% RSLogix 500 project P2_ABIOLA_A_TESTING V7.RSS, saved by version 8.30.00.16 %
PROJECT "UNTITLED"    % processor: Bul.1763 MicroLogix 1100 Series B %

PROGRAM FILES
  LAD 2   4 rungs
  LAD 3 "INPUT DVS"  5 rungs  % This contains all the input devices used %
  LAD 4 "OUTPUT DVS"  4 rungs  % This contains all the output device used %
  LAD 5 "PRO LOGIC"  6 rungs  % This contains the implementation of the logic %

DATA FILES
  O0 OUTPUT  4 elements
  I1 INPUT  6 elements
  S2 STATUS  66 elements
  B3 BINARY  1 elements
  T4 TIMER  2 elements
  C5 COUNTER  1 elements
  R6 CONTROL  1 elements
  N7 INTEGER  1 elements
  F8 FLOAT  1 elements

LADDER 2
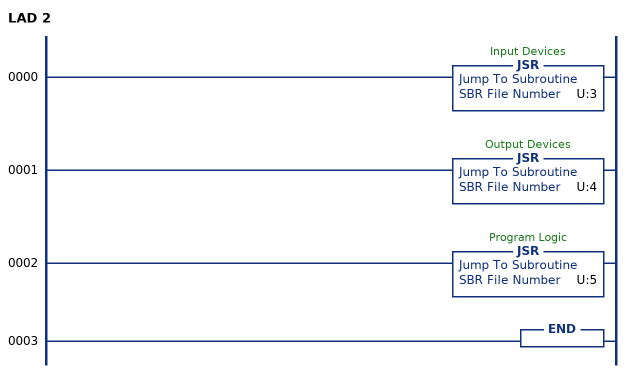
% Rung: 0 %
SOR JSR U:3 EOR
%   U:3  "Input Devices" %
% Rung: 1 %
SOR JSR U:4 EOR
%   U:4  "Output Devices" %
% Rung: 2 %
SOR JSR U:5 EOR
%   U:5  "Program Logic" %
% Rung: 3 %
SOR END EOR

LADDER 3 "INPUT DVS"    % This contains all the input devices used %
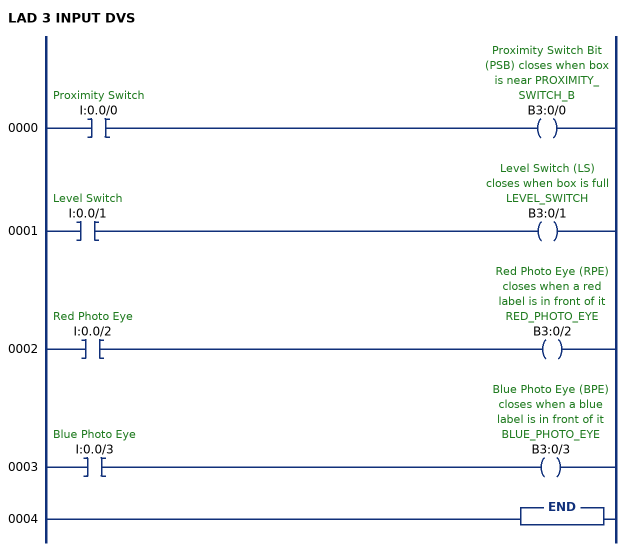
% Rung: 0 %
SOR XIC I:0.0/0 OTE B3:0/0 EOR
%   I:0.0/0  "Proximity Switch" %
%   B3:0/0  PROXIMITY_SWITCH_B  "Proximity Switch Bit (PSB) closes when box is near" %
% Rung: 1 %
SOR XIC I:0.0/1 OTE B3:0/1 EOR
%   I:0.0/1  "Level Switch" %
%   B3:0/1  LEVEL_SWITCH  "Level Switch (LS) closes when box is full" %
% Rung: 2 %
SOR XIC I:0.0/2 OTE B3:0/2 EOR
%   I:0.0/2  "Red Photo Eye" %
%   B3:0/2  RED_PHOTO_EYE  "Red Photo Eye (RPE) closes when a red label is in front of it" %
% Rung: 3 %
SOR XIC I:0.0/3 OTE B3:0/3 EOR
%   I:0.0/3  "Blue Photo Eye" %
%   B3:0/3  BLUE_PHOTO_EYE  "Blue Photo Eye (BPE) closes when a blue label is in front of it" %
% Rung: 4 %
SOR END EOR

LADDER 4 "OUTPUT DVS"    % This contains all the output device used %
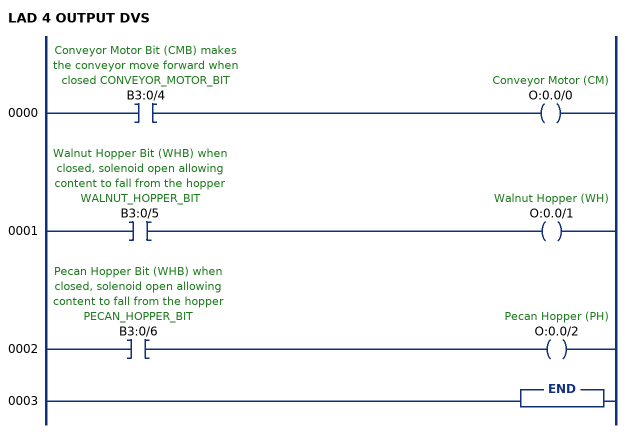
% Rung: 0 %
SOR XIC B3:0/4 OTE O:0.0/0 EOR
%   B3:0/4  CONVEYOR_MOTOR_BIT  "Conveyor Motor Bit (CMB) makes the conveyor move forward when closed" %
%   O:0.0/0  "Conveyor Motor (CM)" %
% Rung: 1 %
SOR XIC B3:0/5 OTE O:0.0/1 EOR
%   B3:0/5  WALNUT_HOPPER_BIT  "Walnut Hopper Bit (WHB) when closed, solenoid open allowing content to fall from the hopper" %
%   O:0.0/1  "Walnut Hopper (WH)" %
% Rung: 2 %
SOR XIC B3:0/6 OTE O:0.0/2 EOR
%   B3:0/6  PECAN_HOPPER_BIT  "Pecan Hopper Bit (WHB) when closed, solenoid open allowing content to fall from the hopper" %
%   O:0.0/2  "Pecan Hopper (PH)" %
% Rung: 3 %
SOR END EOR

LADDER 5 "PRO LOGIC"    % This contains the implementation of the logic %
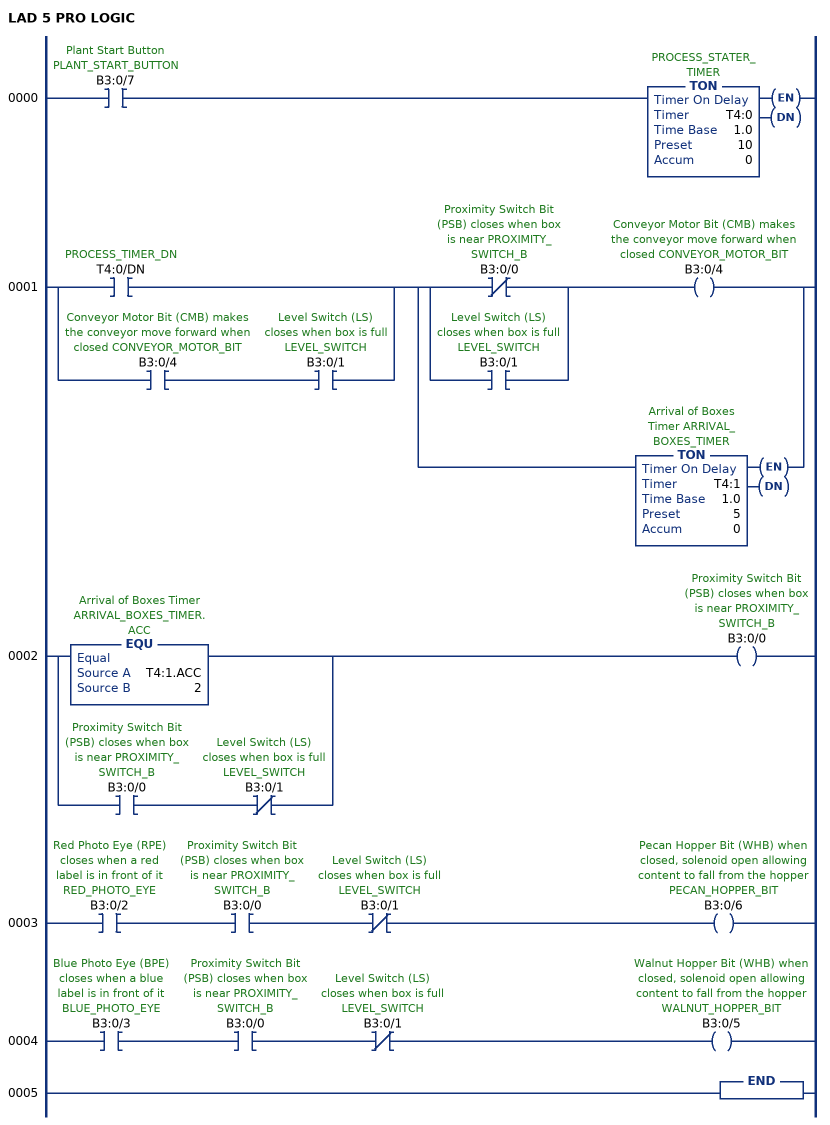
% Rung: 0 %
SOR XIC B3:0/7 TON T4:0 1.0 10 0 EOR
%   B3:0/7  PLANT_START_BUTTON  "Plant Start Button" %
%   T4:0  PROCESS_STATER_TIMER %
% Rung: 1 %
SOR BST XIC T4:0/DN NXB XIC B3:0/4 XIC B3:0/1 BND BST BST XIO B3:0/0 NXB XIC B3:0/1 BND OTE B3:0/4 NXB TON T4:1 1.0 5 0 BND EOR
%   T4:0/DN  PROCESS_TIMER_DN %
%   B3:0/4  CONVEYOR_MOTOR_BIT  "Conveyor Motor Bit (CMB) makes the conveyor move forward when closed" %
%   B3:0/1  LEVEL_SWITCH  "Level Switch (LS) closes when box is full" %
%   B3:0/0  PROXIMITY_SWITCH_B  "Proximity Switch Bit (PSB) closes when box is near" %
%   T4:1  ARRIVAL_BOXES_TIMER  "Arrival of Boxes Timer" %
% Rung: 2 %
SOR BST EQU T4:1.ACC 2 NXB XIC B3:0/0 XIO B3:0/1 BND OTE B3:0/0 EOR
%   T4:1  ARRIVAL_BOXES_TIMER  "Arrival of Boxes Timer" %
%   B3:0/0  PROXIMITY_SWITCH_B  "Proximity Switch Bit (PSB) closes when box is near" %
%   B3:0/1  LEVEL_SWITCH  "Level Switch (LS) closes when box is full" %
% Rung: 3 %
SOR XIC B3:0/2 XIC B3:0/0 XIO B3:0/1 OTE B3:0/6 EOR
%   B3:0/2  RED_PHOTO_EYE  "Red Photo Eye (RPE) closes when a red label is in front of it" %
%   B3:0/0  PROXIMITY_SWITCH_B  "Proximity Switch Bit (PSB) closes when box is near" %
%   B3:0/1  LEVEL_SWITCH  "Level Switch (LS) closes when box is full" %
%   B3:0/6  PECAN_HOPPER_BIT  "Pecan Hopper Bit (WHB) when closed, solenoid open allowing content to fall from the hopper" %
% Rung: 4 %
SOR XIC B3:0/3 XIC B3:0/0 XIO B3:0/1 OTE B3:0/5 EOR
%   B3:0/3  BLUE_PHOTO_EYE  "Blue Photo Eye (BPE) closes when a blue label is in front of it" %
%   B3:0/0  PROXIMITY_SWITCH_B  "Proximity Switch Bit (PSB) closes when box is near" %
%   B3:0/1  LEVEL_SWITCH  "Level Switch (LS) closes when box is full" %
%   B3:0/5  WALNUT_HOPPER_BIT  "Walnut Hopper Bit (WHB) when closed, solenoid open allowing content to fall from the hopper" %
% Rung: 5 %
SOR END EOR

OTHER DOCUMENTED ADDRESSES
  B3:0/8  "One shot"
  B3:0/9  "2 one shot"
  T4:1.PRE  "Arrival of Boxes Comparator"

DATA TABLE (non-zero values as saved)
DATA T4
% .PRE .ACC %
% T4:0 % 10 0
% T4:1 % 5 0
